FUNCTION_BLOCK FB_FieldCodecSint64 IMPLEMENTS I_FieldCodec
VAR_INPUT
END_VAR
VAR_OUTPUT
END_VAR
VAR
    nValue : LINT;
END_VAR

METHOD CalculatePackedDataSize : HRESULT
VAR_INPUT CONSTANT
	anyFirstElem	: T_Any;
	nLength	        : UDINT;        // items to write
END_VAR
VAR_OUTPUT
    nPackedDataSize : UDINT;
END_VAR
VAR
    anyItem         : T_ANY;
    i               : UDINT;
    nValue          : LINT;
END_VAR
anyItem := anyFirstElem;

IF nLength < 1 THEN
    nPackedDataSize := 0;
    RETURN;
END_IF

FOR i := 0  TO nLength - 1 DO
    anyItem.pValue := anyFirstElem.pValue + (i * TO_UDINT(anyFirstElem.diSize)); 
    nValue := PLINT_TO_LINT(anyItem.pValue);
    nPackedDataSize := nPackedDataSize + F_ComputeSInt64Size(nValue);
END_FOR
END_METHOD

METHOD IsPackedRepeatedField : BOOL
VAR_INPUT
	nTag	: UDINT;
END_VAR
IsPackedRepeatedField := F_IsPackedRepeatedField(nTag);
END_METHOD


METHOD ValueReader : HRESULT
VAR_IN_OUT CONSTANT
	aBuffer	: ARRAY [*] OF BYTE;
END_VAR
VAR_IN_OUT
	stState	: ST_ParserInternalState;
END_VAR
VAR_OUTPUT
	anyOut	: T_Any;
END_VAR
VAR 
    nTmp : ULINT;
END_VAR

ValueReader := F_ParseRawVarint64(aBuffer, stState, nTmp);
IF FAILED(ValueReader) THEN
    RETURN;
END_IF
nValue := F_DecodeZigZag64(nTmp);
anyOut := F_ToAnyType(anyArg:= nValue);
END_METHOD

METHOD ValueWriter : HRESULT
VAR_IN_OUT
	aBuffer	: ARRAY [*] OF BYTE;
END_VAR
VAR_IN_OUT
	stState	: ST_WriterInternalState;
END_VAR
VAR_INPUT
    anyIn : T_ANY;
END_VAR
VAR
    nValue  : LINT;
END_VAR

nValue := PLINT_TO_LINT(anyIn.pValue);
ValueWriter := F_WriteSInt64(aBuffer, stState, nValue);
END_METHOD

END_FUNCTION_BLOCK

(* stored: Version 1.1.0.1
   POU FB_FieldCodecSint64: Id {902249f5-4d9a-47d4-8234-bdaacdc871d7}, SpecialFunc None
   Method CalculatePackedDataSize: Id {ce6f6a02-58b9-413d-8739-50e138d454e4}
   Method IsPackedRepeatedField: Id {e7cdeb88-7593-46d4-b96d-f18f55af396f}
   Method ValueReader: Id {b9d1dab2-9dd2-430c-aed8-bbcf1dbe77f8}
   Method ValueWriter: Id {7e533af0-62c5-4ab0-893f-1ea20268bec2} *)
